Fanuc KAREL source: ko00075.KL

-- PROVISIONAL review KL for V1013-1; original PC SHA256 5a2b4d316864929446c7e537a1a098c4a5798391d82544661ec8aba7b3cfdb4b
-- Incomplete behavior may be omitted. Consult companion uncertainty JSON. Do not deploy.
PROGRAM KO00075
%NOLOCKGROUP
BEGIN
  -- UNRESOLVED_PC offsets 5-12; opcodes 9D,23
  -- UNRESOLVED_PC offsets 17-66; opcodes 27,22,1C,27,49,7E,AD,22,31,7E,4A
  -- UNRESOLVED_PC offsets 71-75; opcodes 7F
END KO00075
